(* PLC project Generated.project, CODESYS CODESYS V3.5 SP19 Patch 1 *)
(* stored: creationDateTime 2026-09-14T14:47:22.358308, modificationDateTime 2026-09-14T14:47:22.358308 *)

(* ═══════════════════════════════════════════════════════════════ ↔️ ST_TranslationInterPrg — Bus d'échange inter-PRG produit par PRG_05_Translation ─────────────────────────────────────────────────────────────── 🎯 Rôle : Encapsuler la demande finale M3, l'état public TranslationState et le diagnostic TranslationSafety publiés par PRG_05_Translation vers les consommateurs (PRG_03/06/07). 📤 Producteur unique : PRG_05_Translation (VAR_OUTPUT Data : ST_TranslationInterPrg). 📄 Doc : DOC/AF/AF_Partie-11_Fonction_Translation_v2.3.md 🔌 Architecture : Bus de données typé — encapsulation des échanges inter-PRG. ═══════════════════════════════════════════════════════════════ *)
TYPE ST_TranslationInterPrg : STRUCT
  TranslationFinalInterlockRequest : ST_TranslationFinalInterlockRequest;  (* === ⚡ Demande finale M3 === ↔️ Demande finale et interlocks translation M3 *)
  TranslationState : ST_TranslationState;  (* === 📊 État public translation === 🚦 Etat public translation M3 *)
  TranslationSafety : ST_SafetyTranslation;  (* === 🛡️ Sécurité translation === 🛡️ Diagnostic et securites translation M3 *)
  M3_SensorWordIncoherent : BOOL;  (* === 🎯 Faits decodeur position M3 (produits par PRG_05, AF-02 TBD §8 #5) === ❌ Incoherence detectee mot capteurs M3 *)
  TranslationBusy : BOOL;  (* === ⚙️ États dynamiques & positions stables translation M3 === ⚙️ Translation M3 en mouvement effectif *)
  TranslationDone : BOOL;  (* ✅ Cible translation atteinte et confirmee *)
  M3_AtTremieStable : BOOL;  (* 🎯 M3 positionne stable a la Tremie *)
  M3_AtP1Stable : BOOL;  (* 🎯 M3 positionne stable au Point 1 *)
  M3_AtMaintenanceStable : BOOL;  (* 🎯 M3 positionne stable en zone Maintenance *)
  M3_AtWorkPositionStable : BOOL;  (* 🎯 M3 arrete a une position de travail (P1 ou Maintenance) — STATIQUE (mot capteurs), vrai des le boot sans franchissement. Consomme par le verrou descente treuil T249-A. *)
  TranslationTrace : ST_TraceTranslation;  (* === 🕵️ Trace de blocage terrain (consommée FB_TroubleshootingView) === 🕵️ Trace blocage translation M3 (cause priorisée + horodatage) *)
END_STRUCT;
END_TYPE

(* ═══════════════════════════════════════════════════════════════ 🛡️ ST_SafetyTranslation — Diagnostics de sécurité pour la Translation M3 ─────────────────────────────────────────────────────────────── 🎨 Destiné à l'affichage des défauts de sécurité du translation. ═══════════════════════════════════════════════════════════════ *)
TYPE ST_SafetyTranslation : STRUCT
  Error : BOOL;  (* 🛡️ Bloc sécurité (Safety) en défaut *)
  ErrorId : WORD;  (* ❌ Code bitfield du défaut de sécurité (vue LIVE) *)
  LatchedId : WORD;  (* 🕘 Vue LATCHÉE : ErrorId figé au défaut, effacé au Reset (marqueur [HISTO]) *)
  ErrorOperatorComm : BOOL;  (* 🎮 Perte communication opérateur : joystick CAN ou heartbeat IHM (bit0) *)
  ErrorDriveComm : BOOL;  (* 📡 Perte communication EtherCAT variateur (bit1) *)
  ErrorPhaseRotation : BOOL;  (* ⚡ Mauvaise rotation de phases électriques (bit2) *)
  ErrorBrakeThermal : BOOL;  (* 🌡️ Surchauffe thermique frein commun (bit3) *)
  ErrorMecaB : BOOL;  (* 🛑 Absence confirmation arrêt (Méca B - bit4) *)
  ErrorMecaA : BOOL;  (* 🔄 Mouvement non commandé (Méca A - bit5) *)
  ErrorLimitSwitch : BOOL;  (* 🚧 Limite extrême Translation atteinte (bit6) *)
  ErrorSensorIncoherent : BOOL;  (* 🧭 Mot capteurs M3 incohérent (bit7) *)
  SafeStop : BOOL;  (* 🛡️ Décélération de sécurité demandée *)
  PowerCutOff : BOOL;  (* 🧨 Coupure puissance demandée *)
  EffectivePermitM3_Tremie : BOOL;  (* 🟢 Permis canonique M3 vers Trémie, TRUE = autorisé *)
  EffectivePermitM3_Maintenance : BOOL;  (* 🟢 Permis canonique M3 vers Maintenance/P1, TRUE = autorisé *)
  BlockedBySafety : BOOL;  (* 🚫 Synthèse globale : translation bloquée par la sécurité *)
  PowerCutOffSafety : BOOL;  (* 🧨 Synthèse sécurités critiques entraînant une coupure puissance *)
  SafeStopSafety : BOOL;  (* 🛡️ Synthèse défauts entraînant un SafeStop / Rampe rapide *)
END_STRUCT;
END_TYPE

(* ======================================================================= ↔️ ST_TraceTranslation — Trace de blocage terrain de la translation M3 ─────────────────────────────────────────────────────────────── 🎯 Rôle : Publier au technicien « pourquoi la translation M3 ne bouge pas » : permis de mouvement effectif, interlock hauteur, source SafeStop/coupure et cause de blocage priorisée. 📤 Producteur unique : PRG_05_Translation (Data.TranslationTrace). 📥 Consommateur : FB_TroubleshootingView (pure recopie → GVL_Troubleshooting.S_TraceTranslation). 🔒 Lecture seule — aucun calcul de commande n'en dépend. 🕒 BlockReasonTimestamp : ms depuis démarrage PLC (TIME()), latched au dernier changement de BlockReason (1 scan, mémoire). 📄 Doc métier : DOC/AF/AF_Partie-14_Fonction_Troubleshooting/FB_TroubleshootingView_v1.2.md ======================================================================= *)
TYPE ST_TraceTranslation : STRUCT
  MotionPermitEffective : BOOL;  (* Permis de mouvement effectif (agrégat diagnostic : toutes les barrières levées) 🟢 Translation réellement autorisée à se déplacer *)
  EffectivePermitM3_Tremie : BOOL;  (* Permis directionnels par sens (reflet exact des permis appliqués au mouvement M3) 🟢 Permis canonique M3 vers Trémie (reflet lecture seule) *)
  EffectivePermitM3_Maintenance : BOOL;  (* 🟢 Permis canonique M3 vers Maintenance/P1 (reflet lecture seule) *)
  TremieProcessBlockActive : BOOL;  (* 🛑 Approche trémie interdite par process (trémie pleine / grille levée) — recul libre. Motif du permis trémie rouge. *)
  HeightInterlockBlocking : BOOL;  (* 🚧 Interlock hauteur M1/M2 actif (risque collision) *)
  SafeStopActive : BOOL;  (* Source de blocage — pour distinguer l'origine 🟧 SafeStop effectif appliqué (M3_SafeStop_Aggregate) *)
  SafeStopSourceInput : BOOL;  (* 📥 SafeStop issu du module d'entrée (InputModuleFault) *)
  SafeStopSourceSafety : BOOL;  (* 🛡️ SafeStop issu de FB_Safety_Translation (défaut safety) *)
  PowerCutOffActive : BOOL;  (* 🧨 Coupure puissance amont active *)
  DriveOperational : BOOL;  (* 📡 Variateur AC600 opérationnel *)
  FinalInterlockError : BOOL;  (* Barrière finale (frein / redémarrage) 🛑 Défaut barrière finale (frein / redémarrage) *)
  BlockReason : E_TranslationTraceBlockReason;  (* Cause de blocage priorisée + horodatage 🎯 Cause de blocage prioritaire (ordre de priorité croissant) *)
  BlockReasonTimestamp : UDINT;  (* 🕒 ms depuis démarrage PLC (TIME()) — dernier changement de BlockReason *)
END_STRUCT;
END_TYPE

(* ═══════════════════════════════════════════════════════════════ ↔️ ST_TranslationFinalInterlockRequest — Demande brute vers PDO M3 ─────────────────────────────────────────────────────────────── 📤 Producteur unique : PRG_05_Translation (VAR_OUTPUT). 📥 Consommateur unique : PRG_06_Outputs, avant FB_TranslationOutputInterlock. 🔒 Ne contient jamais une commande PDO autorisée. PowerCutOff : demande safety M3 (FB_Safety_Translation). Consommée par PRG_06_Outputs comme SEULE cause de coupure d'Enable (barrière finale). SafeStop est géré en amont par FB_Translation (rampe rapide, Enable maintenu, AF06 §5). ═══════════════════════════════════════════════════════════════ *)
TYPE ST_TranslationFinalInterlockRequest : STRUCT
  Enable : BOOL;
  Reset : BOOL;
  PowerContactorEngaged : BOOL;
  SafeStop : BOOL;
  EffectivePermitM3_Tremie : BOOL;
  EffectivePermitM3_Maintenance : BOOL;
  PowerCutOff : BOOL;  (* 🧨 Demande coupure puissance (FB_Safety_Translation) — consommée par PRG_06_Outputs (Enable) *)
  BrakeReleaseRequest : BOOL;
  BrakeCommandOpenConfirmed : BOOL;  (* TRUE = contacteur/bobine desserrage confirmé *)
  RequestedDriveControlWord : WORD;  (* 0=None, 1=Fwd, 2=Rev, 7=Reset AC600 *)
  RequestedDriveFreqHz : REAL;
  ReqTremieSemantic : BOOL;  (* TRUE = mouvement demande vers Tremie, independant de InvertDriveDirection *)
  ReqMaintenanceSemantic : BOOL;  (* TRUE = mouvement demande vers Maintenance/P1, independant de InvertDriveDirection *)
END_STRUCT;
END_TYPE

(* ═══════════════════════════════════════════════════════════════ 🚦 ST_TranslationState — États et retours IHM pour la Translation M3 ─────────────────────────────────────────────────────────────── 🎨 Destiné à l'affichage des retours et mesures de la translation M3. ═══════════════════════════════════════════════════════════════ *)
TYPE ST_TranslationState : STRUCT
  FBState : E_State;  (* 🚦 États & diagnostics FB_Translation 🤖 État de l'automate interne (FB_Translation) *)
  AxisBlockReason : E_TranslationTraceBlockReason;  (* 🧩 Cause prioritaire de blocage (miroir de TranslationTrace.BlockReason) *)
  Ready : BOOL;  (* 🟢 Translation prêt à fonctionner *)
  Busy : BOOL;  (* ⚙️ Mouvement en cours *)
  Done : BOOL;  (* ✅ Mouvement terminé avec succès *)
  Error : BOOL;  (* Translation en défaut *)
  ErrorId : WORD;  (* ❌ Code du défaut actif *)
  BrakeCmd : BOOL;  (* 🔓 Commande de desserrage du frein (lecture seule, TRUE = desserré) *)
  BrakeFeedback : BOOL;  (* 🔌 Retour physique direct : TRUE = frein OUVERT (desserré) *)
  PositionSensorTarget : BOOL;  (* 🎯 Capteur de détection de la position cible atteint *)
  PositionReached : BOOL;  (* ✅ Positionneur : cible sélectionnée atteinte (non mémorisé) *)
  DriveActualFreq_Hz : REAL;  (* 📈 Fréquence de sortie réelle du variateur (Hz) *)
  DriveControlWord : WORD;  (* ⚙️ Mot de commande AC600 réellement appliqué *)
  DriveFreqCmd_Hz : REAL;  (* 🎯 Commande fréquence réellement appliquée *)
  ActiveTremie : BOOL;  (* ↔️ Commande active vers Trémie *)
  ActiveMaintenance : BOOL;  (* ↔️ Commande active vers Maintenance *)
  SpeedCmd_Pct : REAL;  (* 📊 Commande active après arbitrage (0.0 à 100.0 %) *)
  FinalInterlockState : E_State;  (* 🛡️ État final lecture seule *)
  FinalInterlockReason : E_TranslationFinalInterlockReason;  (* 🛡️ Cause finale mémorisée *)
  FinalInterlockError : BOOL;  (* 🛡️ Défaut final mémorisé *)
  FinalInterlockErrorId : WORD;  (* 🛡️ Bitfield final *)
  BrakeCommandOpenConfirmed : BOOL;  (* 🔌 Contacteur/bobine desserrage confirmé, pas frein mécanique *)
  FinalBrakeTimeoutElapsed : TIME;  (* ⏱️ Écoulé watchdog 500ms *)
  DriveCommReady : BOOL;  (* 🔌 Diagnostic variateur EtherCAT (décodé — pas de bit-masking côté IHM) 📡 Variateur M3 : communication prête (StatusWord bit7) *)
  DrivePowerReady : BOOL;  (* ⚡ Variateur M3 : puissance prête (StatusWord bit0) *)
  PositionTremie : BOOL;  (* 📍 Mot capteurs et positions Translation M3 *)
  PositionPV : BOOL;
  PositionP2 : BOOL;
  PositionP1 : BOOL;
  PositionMaintenance : BOOL;
  AtTremie : BOOL;  (* : mot EXACT — front franc arrivée/cible (voir PositionXxx ci-dessus = cumulatif zone, réservé ralentissement) jeton "dernier capteur franchi" (front + libération sur mouvement confirmé) — logique de positionnement *)
  AtPV : BOOL;
  AtP2 : BOOL;
  AtP1 : BOOL;
  AtMaintenance : BOOL;
  M3StatusText : STRING(80);  (* T249-B : texte statut position M3 (INFO, lecture seule) — jeton "at position" sur front capteur sinon zone SensorsWord. Ex "M3 a P1 -> Maintenance", "M3 entre P2 et P1" *)
  EstimatedPosM3_M : REAL;  (* 📏 Position continue estimée en mètres (0.0 m Maint -> +X m Trémie) — persistante, survit reboot *)
  SensorsWord : BYTE;  (* bit4=Trémie, bit3=PV, bit2=P2, bit1=P1, bit0=Maintenance *)
  SensorWordIncoherent : BOOL;
  LimitSwitchTremie : BOOL;  (* 🚧 Fin de course extrême Trémie (ex-LimitSwitchFwd) *)
  LimitSwitchMaintenance : BOOL;  (* 🚧 Fin de course extrême Maintenance (ex-LimitSwitchRev) *)
  DriveThermalOk : BOOL;  (* Retour disjoncteur thermique moteur/variateur AC600 — diagnostic seul, l'AC600 se protège lui-même *)
  MaintenanceTargetEnable : BOOL;  (* 🔓 TRUE = Autorise le déplacement vers la cible 4 (Maintenance) ; actif uniquement en mode MAINT_N2 *)
  SimulationModeActive : BOOL;
  HeightInterlockBlocking : BOOL;  (* : TRUE = translation bloquée, M1 ou M2 sous la hauteur mini requise *)
  OdometryGainActive : REAL;  (* 📏 T301 — Odométrie M3 : gain actif + mesure PROPOSÉE P2 <-> PV (jamais appliquée, recopie manuelle) Gain consommé par l'estimateur, m/(Hz.s) *)
  OdometryCalibValid : BOOL;  (* TRUE = gain calculé depuis le réglage Calib* (défaut 2,0 s compris) ; FALSE = gain de repli *)
  OdometryMeasureActive : BOOL;  (* Mesure P2 <-> PV en cours *)
  OdometryMeasuredTime_S : REAL;  (* Dernier temps mesuré P2 <-> PV (s) -> à recopier dans _TranslationCalibTimeP2PV_S *)
  OdometryMeasuredFreqAvg_Hz : REAL;  (* Fréquence moyenne de la mesure (Hz) -> à recopier dans _TranslationCalibFreq_Hz *)
  OdometryMeasuredFreqSpread_Hz : REAL;  (* Écart max - min de fréquence : petit = vitesse constante, mesure fiable *)
  OdometryMeasuredGain : REAL;  (* Gain qui résulterait de la mesure, m/(Hz.s) *)
  OdometryMeasureCount : UDINT;  (* Nombre de mesures abouties depuis le démarrage *)
END_STRUCT;
END_TYPE

(* values of E_TranslationTraceBlockReason: NONE: ✅ Aucun blocage — permis de mouvement effectif; POWER_CUTOFF: 🧨 Coupure puissance amont (instSafetyTranslationM3.PowerCutOff) — priorité max; SAFESTOP: 🟧 SafeStop effectif (InputModule OR safety M3); SAFETY_FAULT: 🛡️ Défaut safety M3 latched (FB_Safety_Translation.Fault.Error); HEIGHT_INTERLOCK: 🚧 Interlock hauteur M1/M2 actif (risque collision); DRIVE_UNAVAILABLE: 📡 Variateur AC600 injoignable / non opérationnel; FINAL_INTERLOCK: 🛑 Barrière finale en défaut (frein / redémarrage); FAULT: ❌ Défaut mouvement M3 latched (FB_Translation.Fault.Error) *)

{attribute 'qualified_only'}
{attribute 'strict'}
TYPE E_TranslationTraceBlockReason : (NONE := 0, POWER_CUTOFF := 1, SAFESTOP := 2, SAFETY_FAULT := 3, HEIGHT_INTERLOCK := 4, DRIVE_UNAVAILABLE := 5, FINAL_INTERLOCK := 6, FAULT := 7);
END_TYPE

(* values of E_State: DISABLED: Enable faux, neutralisé; INIT: Démarrage / vérifs; READY: Prêt, attend ordre; BUSY: Action en cours; DONE: Action terminée; STOPPING: Décél rampe avant arrêt (StartStop=FALSE ou SafeStop=TRUE); ERROR: Défaut actif non acquitté (FB en erreur — HMI non aveugle) *)

{attribute 'qualified_only'}
{attribute 'strict'}
TYPE E_State : (DISABLED := 0, INIT := 1, READY := 2, BUSY := 3, DONE := 4, STOPPING := 5, ERROR := 6);
END_TYPE

{attribute 'qualified_only'}
{attribute 'strict'}
TYPE E_TranslationFinalInterlockReason : (NONE := 0, BRAKE_COMMAND_NOT_CONFIRMED := 1, RESTART_INHIBITED := 2);
END_TYPE
